// TIA Portal V19 export
FUNCTION_BLOCK "Pump_Block"   // FB4, LAD
TITLE = Pump Block
{ S7_Optimized_Access := 'TRUE' }
// Function Block for Pumps
// stored: MemoryReserve 100, SetENOAutomatically false
   VAR_INPUT
      Mode_Selection : Bool;   // Auto or Manual Mode Selected
      Start_Manual : Bool;   // Starting by Manual
      Stop_Manual : Bool;   // Stopping by Manual
      Start_Auto : Bool;   // Starting by Auto
      Stop_Auto : Bool;   // Stopping by Auto
      Level_High : Bool;   // Level High Alarm
      Level_Low : Bool;   // Level Low Alarm
      Set_Time_Start : DInt;   // Setting Timer for Start Auto
      Overload : Bool;   // Motor Overload
      Reset_Fault : Bool;   // Reset Fault Command
   END_VAR
   VAR_OUTPUT
      Pump_Run : Bool;   // Motor Started
      Fault : Bool;   // Motor Fault
      Running_Auto_Mode : Bool;   // Running Auto Mode Signal
   END_VAR
   VAR
      Timer_Start : IEC_TIMER;   // Starting Timer for Auto Mode
      Start_Auto_Activated : Bool;   // Starting Auto Activated
   END_VAR
   VAR_TEMP
      Timer_Start_Output : Bool;   // Output of Timer Started
   END_VAR
   VAR_TEMP   // added for the SCL form of the ladder/FBD networks
      _w1 : Bool;
   END_VAR
BEGIN

REGION Network 1: Motor overload Interlocking
   // If Overloaded trigger a fault
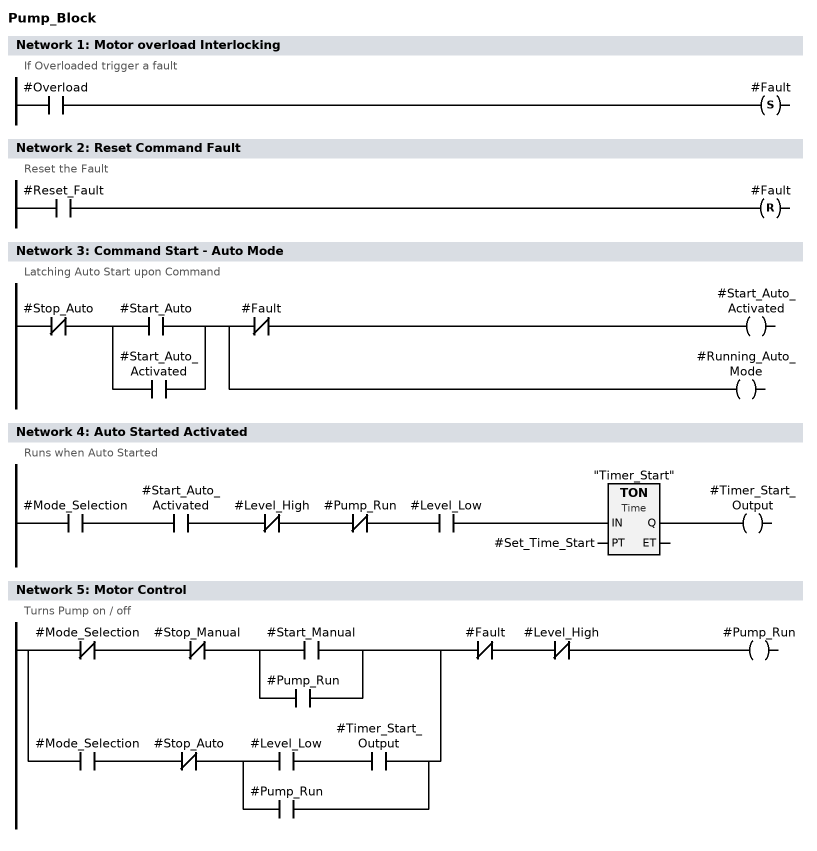
   RUNG wire#powerrail
      Contact( #Overload )
      S_Coil( #Fault )
   END_RUNG
   // the same network as SCL:
   IF #Overload THEN #Fault := TRUE; END_IF;
END_REGION

REGION Network 2: Reset Command Fault
   // Reset the Fault
   RUNG wire#powerrail
      Contact( #Reset_Fault )
      R_Coil( #Fault )
   END_RUNG
   // the same network as SCL:
   IF #Reset_Fault THEN #Fault := FALSE; END_IF;
END_REGION

REGION Network 3: Command Start - Auto Mode
   // Latching Auto Start upon Command
   RUNG wire#powerrail
      I_Contact( #Stop_Auto )
      wire#w1
      Contact( #Start_Auto )
      wire#w2
      I_Contact( #Fault )
      Coil( #Start_Auto_Activated )
   END_RUNG
   RUNG wire#w1
      Contact( #Start_Auto_Activated )
   END_RUNG wire#w2
   RUNG wire#w2
      Coil( #Running_Auto_Mode )
   END_RUNG
   // the same network as SCL:
   #_w1 := NOT #Stop_Auto AND (#Start_Auto OR #Start_Auto_Activated);
   #Start_Auto_Activated := #_w1 AND NOT #Fault;
   #Running_Auto_Mode := #_w1;
END_REGION

REGION Network 4: Auto Started Activated
   // Runs when Auto Started
   RUNG wire#powerrail
      Contact( #Mode_Selection )
      Contact( #Start_Auto_Activated )
      I_Contact( #Level_High )
      I_Contact( #Pump_Run )
      Contact( #Level_Low )
      { S7_Templates := "time_type := Time" } "Timer_Start".TON(pt := #Set_Time_Start, et =>)
      Coil( #Timer_Start_Output )
   END_RUNG
   // the same network as SCL:
   "Timer_Start".TON(IN := #Mode_Selection AND #Start_Auto_Activated AND NOT #Level_High AND NOT #Pump_Run AND #Level_Low,
                     PT := #Set_Time_Start);
   #Timer_Start_Output := "Timer_Start".Q;
END_REGION

REGION Network 5: Motor Control
   // Turns Pump on / off
   RUNG wire#powerrail
      I_Contact( #Mode_Selection )
      I_Contact( #Stop_Manual )
      wire#w1
      Contact( #Start_Manual )
      wire#w2
      I_Contact( #Fault )
      I_Contact( #Level_High )
      Coil( #Pump_Run )
   END_RUNG
   RUNG wire#w1
      Contact( #Pump_Run )
   END_RUNG wire#w2
   RUNG wire#powerrail
      Contact( #Mode_Selection )
      I_Contact( #Stop_Auto )
      wire#w3
      Contact( #Level_Low )
      Contact( #Timer_Start_Output )
   END_RUNG wire#w2
   RUNG wire#w3
      Contact( #Pump_Run )
   END_RUNG wire#w2
   // the same network as SCL:
   #Pump_Run := ((NOT #Mode_Selection AND NOT #Stop_Manual AND (#Start_Manual OR #Pump_Run)) OR (#Mode_Selection AND NOT #Stop_Auto AND ((#Level_Low AND #Timer_Start_Output) OR #Pump_Run))) AND NOT #Fault AND NOT #Level_High;
END_REGION

REGION Network 6: Spare Network
END_REGION
END_FUNCTION_BLOCK
